(* IEC 61131-3 sources: ICSQuartz/benchmarks/oscat_basic_mirror/src, 1 file *)

(* ---- program.st ---- *)
PROGRAM PLC_PRG
VAR_INPUT
    in_STR: STRING;
END_VAR

MIRROR(in_STR);

END_PROGRAM
